INTERFACE ITF_SITP_PolecenieZmiany EXTENDS B_IO.ITF_Przycisk

METHOD PUBLIC ustawStanRozkazu
VAR_INPUT
	bIN				: BOOL;
END_VAR
END_METHOD

(*			
	EVERDE sp. z o.o.
	Rafał Osajda		25.02.2025		TC 4026.13		wer. 0.0.0.1
	Zwraca stan czy rozkaz jest aktywny jeden impuls 
*)
METHOD PUBLIC zwrocStanRozkazu : BOOL
VAR_INPUT
END_VAR
END_METHOD

END_INTERFACE

(* stored: Version 1.1.0.1
   Itf ITF_SITP_PolecenieZmiany: Id {da507f13-6c05-0033-0731-1192d7003616}
   Method ustawStanRozkazu: Id {33101d92-9fd2-0855-21c2-fc1a961fc792}
   Method zwrocStanRozkazu: Id {2ffb1fb4-3ebf-0bf2-06b4-d64cedd67bd1} *)
